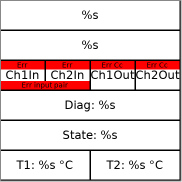
VISUALIZATION TplTsConnectionEK1914  // 182x182
VAR_IN_OUT
	stConnectionDiag 			:FB_TwinSafeConnectionEK1914;
END_VAR
(* End *)
    Rectangle (0,0 180x30), "%s", text variable: stConnectionDiag.sEcSlaveName, colour toggle: stConnectionDiag.sDiag = 'No error'
    Rectangle (0,60 45x30), "Ch1In", colour toggle: stConnectionDiag.bChannel1In
    Rectangle (45,60 45x30), "Ch2In", colour toggle: stConnectionDiag.bChannel2In
    Rectangle (90,60 45x30), "Ch1Out", colour toggle: stConnectionDiag.bChannel1Out
    Rectangle (135,60 45x30), "Ch2Out", colour toggle: stConnectionDiag.bChannel2Out
    Rectangle (0,90 180x30), "Diag: %s", text variable: stConnectionDiag.sDiag, colour toggle: stConnectionDiag.sDiag <> 'No error'
    Rectangle (0,120 180x30), "State: %s", text variable: stConnectionDiag.sState
    Rectangle (0,150 90x30), "T1: %s °C", text variable: stConnectionDiag.stSlaveTemp.nInternalTemperature1, colour toggle: stConnectionDiag.bTempWarning
    Rectangle (90,150 90x30), "T2: %s °C", text variable: stConnectionDiag.stSlaveTemp.nInternalTemperature2, colour toggle: stConnectionDiag.bTempWarning
    Rectangle (0,30 180x30), "%s", text variable: stConnectionDiag.sEcSlaveType
    Rectangle (1,61 43x8), "Err", invisible if: NOT stConnectionDiag.stTsDiagObjectsBitsEK1914.bErrInput1
    Rectangle (46,61 43x8), "Err", invisible if: NOT stConnectionDiag.stTsDiagObjectsBitsEK1914.bErrInput2
    Rectangle (91,61 43x8), "Err Cc", invisible if: NOT stConnectionDiag.stTsDiagObjectsBitsEK1914.bCcErrOutput1
    Rectangle (136,61 43x8), "Err Cc", invisible if: NOT stConnectionDiag.stTsDiagObjectsBitsEK1914.bCcErrOutput2
    Rectangle (1,81 88x8), "Err input pair", invisible if: NOT stConnectionDiag.stTsDiagObjectsBitsEK1914.bErrFirstInputPair
END_VISUALIZATION

(* stored: Version 1.1.0.1, ProductVersion 3.1.4024.11
   Visu TplTsConnectionEK1914: Id {6ff17537-c750-4dee-b381-cf0b20fa7cbc} *)
